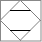
VISUALIZATION VISU_M1Figure_Dryer  // 42x42
    Polygon (40,20) (20,40) (0,20) (20,0)
    Line (10,30) (30,30)
    Line (10,10) (30,10)
END_VISUALIZATION

(* stored: Version 1.1.0.1, ProductVersion 3.1.4019.2
   Visu VISU_M1Figure_Dryer: Id {95799462-05c4-47e1-beaa-72110e9e6f5f} *)
